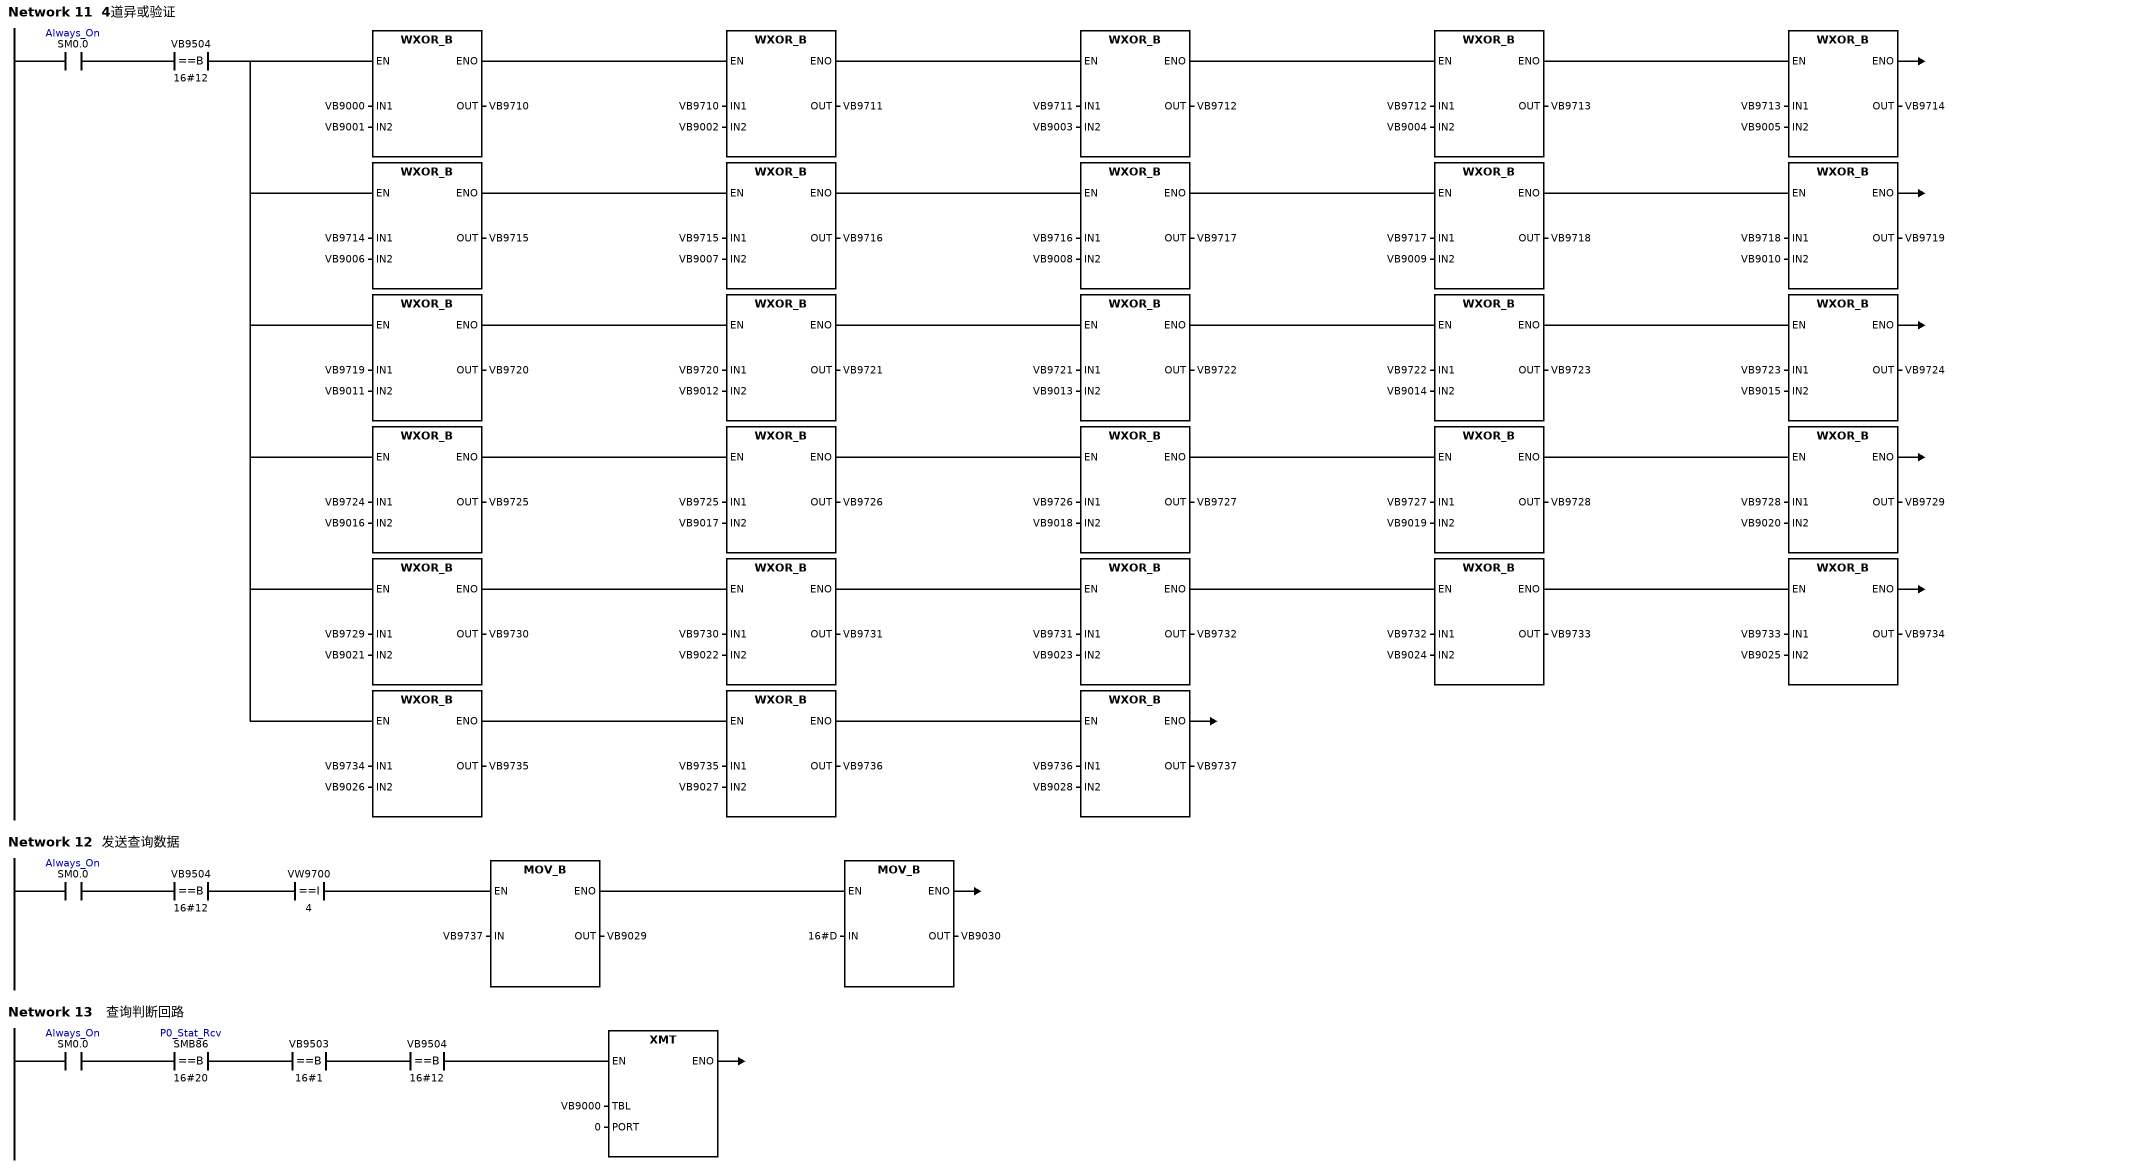
[picture p48: INT1 networks 11-13]
Network 11 // 4道异或验证
LD     Always_On:SM0.0
AB=    VB9504, 16#12
LPS
MOVB   VB9000, VB9710
AENO
XORB   VB9001, VB9710
AENO
MOVB   VB9710, VB9711
AENO
XORB   VB9002, VB9711
AENO
MOVB   VB9711, VB9712
AENO
XORB   VB9003, VB9712
AENO
MOVB   VB9712, VB9713
AENO
XORB   VB9004, VB9713
AENO
MOVB   VB9713, VB9714
XORB   VB9005, VB9714
LRD
MOVB   VB9714, VB9715
AENO
XORB   VB9006, VB9715
AENO
MOVB   VB9715, VB9716
AENO
XORB   VB9007, VB9716
AENO
MOVB   VB9716, VB9717
AENO
XORB   VB9008, VB9717
AENO
MOVB   VB9717, VB9718
AENO
XORB   VB9009, VB9718
AENO
MOVB   VB9718, VB9719
XORB   VB9010, VB9719
LRD
MOVB   VB9719, VB9720
AENO
XORB   VB9011, VB9720
AENO
MOVB   VB9720, VB9721
AENO
XORB   VB9012, VB9721
AENO
MOVB   VB9721, VB9722
AENO
XORB   VB9013, VB9722
AENO
MOVB   VB9722, VB9723
AENO
XORB   VB9014, VB9723
AENO
MOVB   VB9723, VB9724
XORB   VB9015, VB9724
LRD
MOVB   VB9724, VB9725
AENO
XORB   VB9016, VB9725
AENO
MOVB   VB9725, VB9726
AENO
XORB   VB9017, VB9726
AENO
MOVB   VB9726, VB9727
AENO
XORB   VB9018, VB9727
AENO
MOVB   VB9727, VB9728
AENO
XORB   VB9019, VB9728
AENO
MOVB   VB9728, VB9729
XORB   VB9020, VB9729
LRD
MOVB   VB9729, VB9730
AENO
XORB   VB9021, VB9730
AENO
MOVB   VB9730, VB9731
AENO
XORB   VB9022, VB9731
AENO
MOVB   VB9731, VB9732
AENO
XORB   VB9023, VB9732
AENO
MOVB   VB9732, VB9733
AENO
XORB   VB9024, VB9733
AENO
MOVB   VB9733, VB9734
XORB   VB9025, VB9734
LPP
MOVB   VB9734, VB9735
AENO
XORB   VB9026, VB9735
AENO
MOVB   VB9735, VB9736
AENO
XORB   VB9027, VB9736
AENO
MOVB   VB9736, VB9737
XORB   VB9028, VB9737
Network 12 // 发送查询数据
LD     Always_On:SM0.0
AB=    VB9504, 16#12
AW=    VW9700, 4
MOVB   VB9737, VB9029
AENO
MOVB   16#D, VB9030
Network 13 //  查询判断回路
LD     Always_On:SM0.0
AB=    P0_Stat_Rcv:SMB86, 16#20
AB=    VB9503, 16#1
AB=    VB9504, 16#12
XMT    VB9000, 0
END_INTERRUPT_BLOCK
